// Mitsubishi GX Works2 project: 자동차 후진   PLC: Q02/Q02H

PROGRAM MAIN
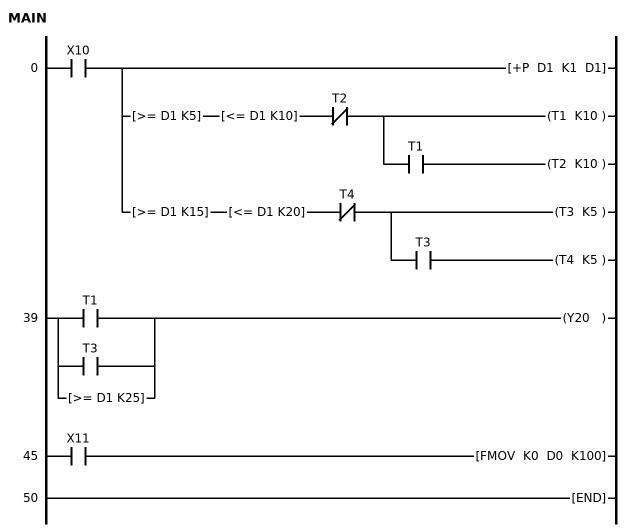
0     LD      X10
      +P      D1 K1 D1
      MPS
      AND>=   D1 K5
      AND<=   D1 K10
      ANI     T2
      OUT     T1 K10
      AND     T1
      OUT     T2 K10
      MPP
      AND>=   D1 K15
      AND<=   D1 K20
      ANI     T4
      OUT     T3 K5
      AND     T3
      OUT     T4 K5
39    LD      T1
      OR      T3
      OR>=    D1 K25
      OUT     Y20
45    LD      X11
      FMOV    K0 D0 K100
50    END
END_PROGRAM
